FUNCTION TriggerCurrentTime : BOOL
VAR_INPUT
END_VAR
VAR
END_VAR
VAR_OUTPUT
	returner: BOOL;
END_VAR


RETURN;

END_FUNCTION

(* stored: Version 1.1.0.1, ProductVersion 3.1.4022.12
   POU TriggerCurrentTime: Id {8bbadcdc-af8c-42f4-bac5-1b3dcc2fd6cd}, SpecialFunc None *)
